// TwinCAT 3 PLC project ScriblyPlc
// ProgramVersion: 3.1.4023.0
// libraries:
//   Tc3_Module,3.3.21.0,Beckhoff Automation GmbH
//   Struckig, 0.9.0.0 (Stefan Besler)
//   ZApplication, 1.3.18.0 (Zeugwerk GmbH)
//   ZAux, 1.3.18.0 (Zeugwerk GmbH)
//   ZCore, 1.3.18.0 (Zeugwerk GmbH)
//   ZEquipment, 1.3.18.0 (Zeugwerk GmbH)
//   ZPlatform, 1.3.18.0 (Zeugwerk GmbH)
// project tree:
//   ZApp/App/ ZApp.TcPOU
//   ZApp/App/_DataTypes/ ZAppStep.TcDUT
//   ZApp/App/_States/ ZAppSequenceBoot.TcPOU, ZAppSequenceBootFault.TcPOU, ZAppSequenceRunning.TcPOU
//   ZApp/App/_SubObjects/ ZAppSequence.TcPOU
//   ZApp/Com/_DataTypes/ ZCom.TcDUT, ZComUnit.TcDUT
//   ZApp/Data/_DataTypes/ ZData.TcDUT, ZDataMachine.TcDUT, ZDataConfig.TcDUT, ZDataCalibration.TcDUT, ZDataRecipe.TcDUT
//   ZApp/Unit/Scribly/ IScribly.TcIO, ScriblyUnit.TcPOU, ScriblyUnitProgram.TcPOU
//   ZApp/Unit/Scribly/Segments/ RingBufferSegment.TcPOU, Segment.TcDUT, SegmentType.TcDUT
//   ZApp/Unit/Scribly/_Com/ ScriblyCom.TcDUT, ScriblyComPublish.TcDUT, ScriblyComPublishEquipment.TcDUT, ScriblyComRef.TcDUT, ScriblyComRequest.TcDUT, ScriblyComSubscribe.TcDUT, ScriblyComSubscribeEquipment.TcDUT, ScriblyComSubscribeSegments.TcDUT
//   ZApp/Unit/Scribly/_DataTypes/ ScriblyState.TcDUT, ScriblyStep.TcDUT
//   ZApp/Unit/Scribly/_Data/ ScriblyDataCalibration.TcDUT, ScriblyDataConfig.TcDUT, ScriblyDataMachine.TcDUT, ScriblyDataRef.TcDUT
//   ZApp/Unit/Scribly/_Equipment/ ScriblyActuator.TcPOU, ScriblyActuatorPen.TcPOU, ScriblyAxis.TcPOU, ScriblyEquipment.TcPOU, ScriblyFieldbus.TcPOU, ScriblyIo.TcPOU, ScriblyLinkedUnit.TcPOU
//   ZApp/Unit/Scribly/_States/ ScriblySequenceAutomatic.TcPOU, ScriblySequenceBoot.TcPOU, ScriblySequenceFaultReaction.TcPOU, ScriblySequenceGoHome.TcPOU, ScriblySequenceStop.TcPOU
//   ZApp/Unit/Scribly/_SubObjects/ ScriblyContainer.TcPOU, ScriblySequence.TcPOU
//   ZApp/ ZGlobal.TcGVL, ZModuleProgram.TcPOU, ZModuleTask.TcTTO
// real-time tasks:
//   TASK ZModuleTask: cycle T#10ms, priority 20, ADS port 350

CONFIGURATION ScriblyPlc
    RESOURCE PLC ON TwinCAT3
        TASK ZModuleTask(INTERVAL := T#10ms, PRIORITY := 20);
        PROGRAM ZeugwerkFramework WITH ZModuleTask : ZeugwerkFramework;
        PROGRAM ZModuleProgram WITH ZModuleTask : ZModuleProgram;
    END_RESOURCE
END_CONFIGURATION

// ---- ZApp/App/_DataTypes/ZAppStep.TcDUT
{attribute 'qualified_only'}
{attribute 'to_string'}
TYPE ZAppStep :
(
  Undefined := 0
  
  ,BootBegin
  ,BootLoadDefaultData
  ,BootEnd
  ,BootFaultBegin
  ,BootFaultEnd 
  ,RunningBegin
  ,RunningEnd   
);
END_TYPE

// ---- ZApp/Com/_DataTypes/ZCom.TcDUT
TYPE ZCom :
STRUCT
  // module context
  App : ZApplication.ApplicationComPublish;
  Alarming : ZApplication.AlarmingCom;
  Messages : ZApplication.MessagingCom;
  
  // unit context
  Unit : ZComUnit;

END_STRUCT
END_TYPE

// ---- ZApp/Com/_DataTypes/ZComUnit.TcDUT
TYPE ZComUnit :
STRUCT
{region "Scribly"}
{IF NOT (defined (Scribly_disabled))}
  Scribly : ScriblyCom;
  {attribute 'ZId' := '61e5b130-0fef-4d8b-85dd-afb1efcde47c'}
{END_IF}
{endregion}
{attribute '__ZwPlcApplicationComUnitDeclaration__'} // Do not remove this attribute! It is used for code generation.
END_STRUCT
END_TYPE

// ---- ZApp/Data/_DataTypes/ZData.TcDUT
TYPE ZData :
STRUCT
  Config : ZDataConfig;
  Machine : ZDataMachine;
  Calibration : ZDataCalibration;
  Recipe : ZDataRecipe;
END_STRUCT
END_TYPE

// ---- ZApp/Data/_DataTypes/ZDataMachine.TcDUT
TYPE ZDataMachine :
STRUCT
{region "Scribly"}
{IF NOT (defined (Scribly_disabled))}
  Scribly : ScriblyDataMachine;
  {attribute 'ZId' := '61e5b130-0fef-4d8b-85dd-afb1efcde47c'}
{END_IF}
{endregion}
{attribute '__ZwPlcApplicationDataMachineDeclaration__'} // Do not remove this attribute! It is used for code generation.
END_STRUCT
END_TYPE

// ---- ZApp/Data/_DataTypes/ZDataConfig.TcDUT
TYPE ZDataConfig :
STRUCT
{region "Scribly"}
{IF NOT (defined (Scribly_disabled))}
  Scribly : ScriblyDataConfig;
  {attribute 'ZId' := '61e5b130-0fef-4d8b-85dd-afb1efcde47c'}
{END_IF}
{endregion}
{attribute '__ZwPlcApplicationDataConfigDeclaration__'} // Do not remove this attribute! It is used for code generation.
END_STRUCT
END_TYPE

// ---- ZApp/Data/_DataTypes/ZDataCalibration.TcDUT
TYPE ZDataCalibration :
STRUCT
{region "Scribly"}
{IF NOT (defined (Scribly_disabled))}
  Scribly : ScriblyDataCalibration;
  {attribute 'ZId' := '61e5b130-0fef-4d8b-85dd-afb1efcde47c'}
{END_IF}
{endregion}
{attribute '__ZwPlcApplicationDataCalibrationDeclaration__'} // Do not remove this attribute! It is used for code generation.
END_STRUCT
END_TYPE

// ---- ZApp/Data/_DataTypes/ZDataRecipe.TcDUT
TYPE ZDataRecipe :
STRUCT
  RecipeParam1 : LREAL;
  RecipeParam2 : LREAL;
  RecipeParam3 : LREAL;
END_STRUCT
END_TYPE

// ---- ZApp/Unit/Scribly/Segments/Segment.TcDUT
TYPE Segment :
STRUCT
  Verb : SegmentType;
  Points : ARRAY[0..7] OF ZCore.Vector4;
END_STRUCT
END_TYPE

// ---- ZApp/Unit/Scribly/Segments/SegmentType.TcDUT
{attribute 'qualified_only'}
{attribute 'strict'}
TYPE SegmentType :
(
	Location := 0,
  LinePoints,
  CatmulRomPoints
);
END_TYPE

// ---- ZApp/Unit/Scribly/_Com/ScriblyCom.TcDUT
/// This struct contains variables that
/// * are read from outside (e.g. HMI) to retrieve information about the unit's current state and (temporary) parameters (= `publish`) 
/// * are written from outside (e.g. HMI) to control the unit via ADS (= `subscribe`) 
TYPE ScriblyCom :
STRUCT
  Publish : ScriblyComPublish;
  Subscribe : ScriblyComSubscribe;
END_STRUCT
END_TYPE

// ---- ZApp/Unit/Scribly/_Com/ScriblyComPublish.TcDUT
/// this is the container of informations that the unit wants to share with the world outside of the PLC
/// This struct should only be read from by external applications.
TYPE ScriblyComPublish :
STRUCT
  State : ZApplication.UnitStateMachineState; // state the unit is in
  Request : ScriblyComRequest; // booleans that indictate which action is currently possible to perform with this unit
  Equipment : ScriblyComPublishEquipment;  // structs for equipment objects which are used by the bridges
END_STRUCT
END_TYPE

// ---- ZApp/Unit/Scribly/_Com/ScriblyComPublishEquipment.TcDUT
TYPE ScriblyComPublishEquipment :
STRUCT

{region "Pen : ActuatorDigital"}
  Pen : ZApplication.ActuatorDigitalComPublish;
  PenDown : ZApplication.DigitalComPublish;
  PenUp : ZApplication.DigitalComPublish;
  PenIsDown : ZApplication.DigitalComPublish;
  PenIsUp : ZApplication.DigitalComPublish;
  {attribute 'ZId' := '715ceec0-4c65-4cb8-884b-f54d8c494ea5'}
{endregion}

{region "AxisX : Axis"}
  AxisX : ZApplication.AxisComPublish;
  {attribute 'ZId' := 'a9303431-20fb-4f90-9643-84006bcd2555'}
{endregion}

{region "AxisY : Axis"}
  AxisY : ZApplication.AxisComPublish;
  {attribute 'ZId' := '787e5d02-9d93-4b03-8235-ee23b1a291ad'}
{endregion}

{attribute '__ZwPlcUnitComDeclaration__'} // Do not remove this attribute! It is used for code generation.

END_STRUCT
END_TYPE

// ---- ZApp/Unit/Scribly/_Com/ScriblyComRef.TcDUT
/// container for all communication data types that are used by the unit
TYPE ScriblyComRef :
STRUCT
  Publish : REFERENCE TO ScriblyComPublish; 
  Subscribe : REFERENCE TO ScriblyComSubscribe; 
END_STRUCT
END_TYPE

// ---- ZApp/Unit/Scribly/_Com/ScriblyComRequest.TcDUT
TYPE ScriblyComRequest :
STRUCT
  Start : BOOL;
  Stop : BOOL;
  GoHome : BOOL;
  Halt : BOOL;
END_STRUCT
END_TYPE

// ---- ZApp/Unit/Scribly/_Com/ScriblyComSubscribe.TcDUT
TYPE ScriblyComSubscribe :
STRUCT
  Request : ScriblyComRequest; // contains booleans that are used to start a specific sequence.
  Equipment : ScriblyComSubscribeEquipment;  // structs for equipment objects which are used by the bridges
  
  Segments : ScriblyComSubscribeSegments;
END_STRUCT
END_TYPE

// ---- ZApp/Unit/Scribly/_Com/ScriblyComSubscribeEquipment.TcDUT
TYPE ScriblyComSubscribeEquipment :
STRUCT

{region "Pen : ActuatorDigital"}
  Pen : ZApplication.ActuatorDigitalComSubscribe;
  PenDown : ZApplication.DigitalComSubscribe;
  PenUp : ZApplication.DigitalComSubscribe;
  PenIsDown : ZApplication.DigitalComSubscribe;
  PenIsUp : ZApplication.DigitalComSubscribe;
  {attribute 'ZId' := '715ceec0-4c65-4cb8-884b-f54d8c494ea5'}
{endregion}

{region "AxisX : Axis"}
  AxisX : ZApplication.AxisComSubscribe;
  {attribute 'ZId' := 'a9303431-20fb-4f90-9643-84006bcd2555'}
{endregion}

{region "AxisY : Axis"}
  AxisY : ZApplication.AxisComSubscribe;
  {attribute 'ZId' := '787e5d02-9d93-4b03-8235-ee23b1a291ad'}
{endregion}

{attribute '__ZwPlcUnitComDeclaration__'} // Do not remove this attribute! It is used for code generation.

END_STRUCT
END_TYPE

// ---- ZApp/Unit/Scribly/_Com/ScriblyComSubscribeSegments.TcDUT
TYPE ScriblyComSubscribeSegments :
STRUCT
  Start : DINT;
  End : DINT;
  Data : ARRAY[0..10] OF Segment;
END_STRUCT
END_TYPE

// ---- ZApp/Unit/Scribly/_DataTypes/ScriblyState.TcDUT
/// This enumeration contains all used defined sequences of a unit.
/// Per default a unit makes use of the states that are contained in (UnitStateDefault)[xref:ZApplication.UnitStateDefault]. However,
/// most of the time a unit need to perform some application depend sequences that can be performed by putting the unit into userdefined states.
/// For instance, a robotic unit could use the state (automatic)[xref:ZApplication.UnitStateDefault] to lift an object from point A to point B,
/// a userdefined state could be used to open and close the robotic-units gripper, respectively
{attribute 'qualified_only'}
TYPE ScriblyState :
(
	UserdefinedState1 := ZApplication.UnitStateMachineState.Last+1
);
END_TYPE

// ---- ZApp/Unit/Scribly/_DataTypes/ScriblyStep.TcDUT
/// This enumeration contains all steps that are used by the various sequences of a unit.
/// Sequences use a subrange (***Begin to ***End) of this enumeration.
{attribute 'qualified_only'}
{attribute 'to_string'}
TYPE ScriblyStep :
(
  Undefined := 0
  
  ,BootBegin
  ,BootEnd 

  ,StopBegin
  ,StopEnd

  ,AutomaticBegin
  ,AutomaticWaitSegment
  ,AutomaticMoveToSegmentStart
  ,AutomaticMovePenDown
  ,AutomaticDraw
  ,AutomaticMovePenUp
  ,AutomaticDrawLine
  ,AutomaticDrawCatmulRomDrawSplineBegin
  ,AutomaticDrawCatmulRomDrawSpline
  ,AutomaticEnd
  
  ,GoHomeBegin
  ,GoHomeMoveUp  
  ,GoHomeReferenceXY
  ,GoHomeEnd 
  
  ,FaultReactionBegin
  ,FaultReactionEnd
);
END_TYPE

// ---- ZApp/Unit/Scribly/_Data/ScriblyDataCalibration.TcDUT
/// calibration that is determined by calibration sequences of the unit (static offsets, shifts)
TYPE ScriblyDataCalibration :
STRUCT
END_STRUCT
END_TYPE

// ---- ZApp/Unit/Scribly/_Data/ScriblyDataConfig.TcDUT
/// configuration data that is used during boot to configure the Units equipment
TYPE ScriblyDataConfig :
STRUCT
  Simulated : BOOL;
END_STRUCT
END_TYPE

// ---- ZApp/Unit/Scribly/_Data/ScriblyDataMachine.TcDUT
/// machine data that is used through most sequences of the unit (motor speed, axes positions, ...)
TYPE ScriblyDataMachine :
STRUCT
  Slowspeed : LREAL;
  Highspeed : LREAL;
END_STRUCT
END_TYPE

// ---- ZApp/Unit/Scribly/_Data/ScriblyDataRef.TcDUT
/// container for all data that are used by the unit
TYPE ScriblyDataRef :
STRUCT
  Config : REFERENCE TO ScriblyDataConfig; // data required for booting the unit (axes configuration, simulation, parameters that have to be written in PREOP, ...)
  Machine : REFERENCE TO ScriblyDataMachine; // speeds, positions, ...
  Calibration : REFERENCE TO ScriblyDataCalibration; // offsets, shifts of nominal to actual values
END_STRUCT
END_TYPE

// ---- ZApp/ZGlobal.TcGVL
{attribute 'qualified_only'}
VAR_GLOBAL
  Com : ZCom;
END_VAR
VAR_GLOBAL PERSISTENT
  Data : ZData;
END_VAR

// ---- ZApp/Unit/Scribly/IScribly.TcIO
INTERFACE IScribly EXTENDS ZApplication.IUnit

END_INTERFACE

// ---- ZApp/ZModuleProgram.TcPOU
/// Zeugwerk Application
PROGRAM ZModuleProgram
VAR
{region "ZModuleProgram : Utility"}
  App : ZApp(name:='Scribly', com:=ZGlobal.Com.App);
  Datetime : ZAux.DateTimeUM;
  {attribute 'ZId' := ''}
{endregion}
{region "ZModuleProgram : Logging"}
  Alarming : ZApplication.Alarming(App, datetime := Datetime, com := ZGlobal.Com.Alarming);
  LoggerHmi : ZApplication.Messaging(App, datetime := Datetime, com := ZGlobal.Com.Messages);
  LoggerFile : ZAux.LoggerFile7FF(App, datetime := Datetime, filePath:='C:\Zeugwerk\logs\messages.log', target:='');
  Logger : ZAux.Logging;
  {attribute 'ZId' := ''}
{endregion}  
{attribute '__ZwPlcApplicationModuleProgramDeclaration__'} // Do not remove this attribute! It is used for code generation.
{region "Scribly"}
{undefine RunInSeparateProgram}
{IF NOT (defined (Scribly_disabled)) AND NOT (defined (RunInSeparateProgram))}
  Scribly : ScriblyUnit(name := 'Scribly', // name of the unit (for logging)
					  parent := App, // caller of the Unit's cyclic method. If the Unit runs in its own context use 0
						configdata := ZGlobal.Data.Config.Scribly,
						machinedata := ZGlobal.Data.Machine.Scribly,
						calibrationdata := ZGlobal.Data.Calibration.Scribly,
						com := ZGlobal.Com.Unit.Scribly);
  {attribute 'section' := '__ZwPlcUnitProgramDeclaration__'}
  {attribute 'ZId' := '61e5b130-0fef-4d8b-85dd-afb1efcde47c'}
{END_IF}
{endregion}
{attribute '__ZwPlcUnitProgramDeclaration__'} // Do not remove this attribute! It is used for code generation.
END_VAR

{region "ZModuleProgram : Utility"}
  Datetime.Cyclic();
  App.Cyclic();
  {attribute 'ZId' := ''}
{endregion}
{attribute '__ZwPlcApplicationModuleProgramImplementation__'} // Do not remove this attribute! It is used for code generation.

END_PROGRAM

// ---- ZApp/App/ZApp.TcPOU
FUNCTION_BLOCK ZApp EXTENDS ZApplication.Application
VAR
  _boot : ZAppSequenceBoot;
  _bootFault : ZAppSequenceBootFault;
  _running : ZAppSequenceRunning;
END_VAR

METHOD FB_init : BOOL
VAR_INPUT
  bInitRetains : BOOL; /// if TRUE, the retain variables are initialized (warm start / cold start)
  bInCopyCode : BOOL; /// if TRUE, the instance afterwards gets moved into the copy code (online change)
  name : ZCore.ZString;
  com : REFERENCE TO ZApplication.ApplicationComPublish;
END_VAR
SetBootSequence(_boot);
SetBootFaultSequence(_bootFault);
SetRunningSequence(_running);
END_METHOD

END_FUNCTION_BLOCK

// ---- ZApp/App/_States/ZAppSequenceBoot.TcPOU
FUNCTION_BLOCK ZAppSequenceBoot EXTENDS ZAppSequence IMPLEMENTS ZCore.ISequence
VAR
  _step : ZCore.Step(ZAppStep.BootBegin, ZAppStep.BootEnd);
END_VAR

IF OnStart(_step)
THEN
  // init custom sequence variables here ...
END_IF

REPEAT
  LogStep();

  CASE _step.Index OF
    (* -------------------------------------------------------------------------------------------------------------------------------- *)
    ZAppStep.BootBegin:
    (* -------------------------------------------------------------------------------------------------------------------------------- *)
    
      IF _step.OnEntry()
      THEN
        ZModuleProgram.LoggerFile.SetLevel(ZCore.LogLevel.Trace);
        ZModuleProgram.Logger.AddLogger(ZModuleProgram.LoggerFile);        
        {attribute '__ZwPlcAppZComModuleContext__'} // Do not remove this attribute! It is used for code generation.      
      END_IF
      
	  IF ZModuleProgram.Datetime.State <> ZCore.ObjectState.Booting
      THEN
        _step.SetNext(ZAppStep.BootLoadDefaultData);        
      END_IF
      
    (* -------------------------------------------------------------------------------------------------------------------------------- *)
    ZAppStep.BootLoadDefaultData:
    (* -------------------------------------------------------------------------------------------------------------------------------- *)

      {warning 'The application is loading the default config data on every restart!'}
      LoadDefaultConfigData();
      
      IF IsCommissioning()
      THEN
        LoadDefaultData();
      END_IF
      
      _step.SetNext(ZAppStep.BootEnd);
      
    (* -------------------------------------------------------------------------------------------------------------------------------- *)
    ZAppStep.BootEnd:
    (* -------------------------------------------------------------------------------------------------------------------------------- *)
      SetBusy(FALSE);
      
  ELSE
    Abort('sequence contains unhandled step');
  END_CASE
UNTIL _step.IsNotRepeatable() OR_ELSE NOT Busy END_REPEAT

METHOD  IsCommissioning : BOOL
IsCommissioning := TRUE;
END_METHOD

METHOD FINAL LoadDefaultConfigData

{region "Scribly"}
  {IF NOT (defined (Scribly_disabled))}
  ZGlobal.Data.Config.Scribly.Simulated := TRUE;
  {region "UserInitCode"}
  // put your individual init code for this unit here
  {endregion}
  {END_IF}
  {attribute 'ZId' := '61e5b130-0fef-4d8b-85dd-afb1efcde47c'}
{endregion}

{attribute '__ZwPlcUnitLoadDefaultConfigData__'} // Do not remove this attribute! It is used for code generation.
END_METHOD

METHOD FINAL LoadDefaultData

{attribute '__ZwPlcUnitLoadDefaultData__'} // Do not remove this attribute! It is used for code generation.
ZGlobal.Data.Machine.Scribly.Highspeed := 100;
ZGlobal.Data.Machine.Scribly.Slowspeed := 10;
END_METHOD

END_FUNCTION_BLOCK

// ---- ZApp/App/_SubObjects/ZAppSequence.TcPOU
FUNCTION_BLOCK ABSTRACT ZAppSequence EXTENDS ZApplication.Sequence IMPLEMENTS ZCore.ISequence

METHOD StepDecoded : ZCore.ZString
VAR_INPUT
  stepIndex : INT;
END_VAR
VAR_INST
  _stepIndexDecoded : ZAppStep;
END_VAR
_stepIndexDecoded := stepIndex;
StepDecoded := TO_STRING(_stepIndexDecoded);
END_METHOD

END_FUNCTION_BLOCK

// ---- ZApp/App/_States/ZAppSequenceBootFault.TcPOU
FUNCTION_BLOCK ZAppSequenceBootFault EXTENDS ZAppSequence IMPLEMENTS ZCore.ISequence
VAR
  _step : ZCore.Step(ZAppStep.BootFaultBegin, ZAppStep.BootFaultEnd);
END_VAR

IF OnStart(_step)
THEN
  // init custom sequence variables here ...
END_IF

REPEAT
  LogStep();

  CASE _step.Index OF
    (* -------------------------------------------------------------------------------------------------------------------------------- *)
    ZAppStep.BootFaultBegin:
    (* -------------------------------------------------------------------------------------------------------------------------------- *)
      _step.SetNext(ZAppStep.BootFaultEnd);
      
    (* -------------------------------------------------------------------------------------------------------------------------------- *)
    ZAppStep.BootFaultEnd:
    (* -------------------------------------------------------------------------------------------------------------------------------- *)
      SetBusy(FALSE);
      
  ELSE
    Abort('sequence contains unhandled step');
  END_CASE
UNTIL _step.IsNotRepeatable() OR_ELSE NOT Busy END_REPEAT

END_FUNCTION_BLOCK

// ---- ZApp/App/_States/ZAppSequenceRunning.TcPOU
FUNCTION_BLOCK ZAppSequenceRunning EXTENDS ZAppSequence IMPLEMENTS ZCore.ISequence
VAR
  _step : ZCore.Step(ZAppStep.RunningBegin, ZAppStep.RunningEnd);
END_VAR

IF OnStart(_step)
THEN
  // init custom sequence variables here ...
END_IF

REPEAT
  LogStep();

  CASE _step.Index OF
    (* -------------------------------------------------------------------------------------------------------------------------------- *)
    ZAppStep.RunningBegin:
    (* -------------------------------------------------------------------------------------------------------------------------------- *)
      ; // implement me
      
    (* -------------------------------------------------------------------------------------------------------------------------------- *)
    ZAppStep.RunningEnd:
    (* -------------------------------------------------------------------------------------------------------------------------------- *)
      SetBusy(FALSE);
      
  ELSE
    Abort('sequence contains unhandled step');
  END_CASE
UNTIL _step.IsNotRepeatable() OR_ELSE NOT Busy END_REPEAT

END_FUNCTION_BLOCK

// ---- ZApp/Unit/Scribly/ScriblyUnit.TcPOU
/// Declaration of a distinct unit of this application
FUNCTION_BLOCK ScriblyUnit EXTENDS ZApplication.Unit IMPLEMENTS IScribly, ZAux.IStateMachineListener
VAR
  _equipment : ScriblyEquipment(THIS^);
  _data : ScriblyDataRef;
  _com : ScriblyComRef;

  _boot : ScriblySequenceBoot(THIS^);
  _automatic : ScriblySequenceAutomatic(THIS^);
  _stop : ScriblySequenceStop(THIS^);
  _gohome : ScriblySequenceGoHome(THIS^);
  _faultReaction : ScriblySequenceFaultReaction(THIS^);
  
  _statemachine : ZApplication.UnitStateMachine;

  _observeTimer : ZAux.Timer;
  _segments : RingBufferSegment(
                10, 
                ADR(ZGlobal.Com.Unit.Scribly.Subscribe.Segments.Start),
                ADR(ZGlobal.Com.Unit.Scribly.Subscribe.Segments.End),
                ADR(ZGlobal.Com.Unit.Scribly.Subscribe.Segments.Data));        
END_VAR

{attribute 'ZId' := 'f607484c-b594-4144-a307-86b8991e3218'}

IF _observeTimer.Done THEN
  _observeTimer.WaitAsync(0.1);
  
  // monitor _com for requested actions (e.g. start homing, start automatic mode, ...)
  ObserveRequest(_com.Subscribe.Request.Start, ZApplication.UnitStateMachineState.Automatic);
  ObserveRequest(_com.Subscribe.Request.Stop, ZApplication.UnitStateMachineState.Stop);
  ObserveRequest(_com.Subscribe.Request.GoHome, ZApplication.UnitStateMachineState.GoHome);
  ObserveRequest(_com.Subscribe.Request.Halt, ZApplication.UnitStateMachineState.Halt);
  
  // provide relevant information via ADS
  _com.Publish.Request.Stop := _stateMachine.IsTransitionAllowed(ZApplication.UnitStateMachineState.Stop);
  _com.Publish.Request.Start := _stateMachine.IsTransitionAllowed(ZApplication.UnitStateMachineState.Automatic);
  _com.Publish.Request.GoHome := _stateMachine.IsTransitionAllowed(ZApplication.UnitStateMachineState.GoHome);
  _com.Publish.Request.Halt := _stateMachine.IsTransitionAllowed(ZApplication.UnitStateMachineState.Halt);

  _com.Publish.State := _stateMachine.State();
END_IF

METHOD FB_init : BOOL
VAR_INPUT
  bInitRetains : BOOL; // if TRUE, the retain variables are initialized (warm start / cold start)
  bInCopyCode : BOOL;  // if TRUE, the instance afterwards gets moved into the copy code (online change)
  parent : ZCore.IManagedObject; // caller of the Unit's cyclic method. If the Unit runs in its own context use 0
  name : ZCore.ZString;  // name of this unit as it should show up in the logger
  configdata : REFERENCE TO ScriblyDataConfig;  // reference to the configuration data that is used during boot to configure the Units equipment
  machinedata : REFERENCE TO ScriblyDataMachine; // reference to the machine data that is used through most sequences of the unit (motor speed, axes positions, ...)
  calibrationdata : REFERENCE TO ScriblyDataCalibration;  // reference to calibration that is determined by calibration sequences of the unit (static offsets, shifts)
  com : REFERENCE TO ScriblyCom;  // reference to the communication interface that is used to control this Unit via ADS
END_VAR
_name := name;

// initialize local logger decorator
_loggerDecorator.FB_init(bInitRetains, bInCopyCode, name, ZModuleProgram.Logger);
_alarmingDecorator.FB_init(bInitRetains, bInCopyCode, name, ZModuleProgram.Alarming);

// setup data
_data.Config REF= configdata;
_data.Machine REF= machinedata;
_data.Calibration REF= calibrationdata;
_com.Publish REF= com.Publish;
_com.Subscribe REF= com.Subscribe;

// ------- sequence initialization, map sequences of this unit to the statemachine -------
{attribute '__ZwPlcUnitInitSequenceImplementation__'} // Do not remove this attribute! It is used for code generation.
_statemachine.SetSequence(ZApplication.UnitStateMachineState.Boot, _boot);
_statemachine.SetSequence(ZApplication.UnitStateMachineState.FaultReaction, _faultReaction);
_statemachine.SetSequence(ZApplication.UnitStateMachineState.Gohome, _gohome);
_statemachine.SetSequence(ZApplication.UnitStateMachineState.Stop, _stop);
_statemachine.SetSequence(ZApplication.UnitStateMachineState.Automatic, _automatic);

_statemachine.SetName(_name);
_statemachine.SetListener(THIS^);
_statemachine.SetLogger(_logger);

// set initial state
_statemachine.SetState(ZApplication.UnitStateMachineState.Boot);
_statemachineIntrf := _statemachine;
END_METHOD

/// This method is called by a [Statemachine's startTransition method](xref:ZApplication.UnitStateMachine#startTransition)
/// if a given transition was failed (e.g. the transition is not allowed according to the state diagram of the state machine).
/// The State that was active previously in the StateMachine remains active and `requestedState` indicates which state transition
/// was requested by the user.
METHOD OnStartTransitionFailed
VAR_INPUT
  state : INT;  
  requestedState : INT;
END_VAR
END_METHOD

/// This method is called by a [Statemachine's startTransition method](xref:ZApplication.UnitStateMachine#startTransition)
/// if a given transition was successful. Please note, that at the time this event occurs, `state` still holds the
/// state that was active before calling `startTransition`, there is still one more call to this `state` to allow it to 
/// cleanup.
METHOD OnStartTransitionSucceeded
VAR_INPUT
  state : INT;  
  newState : INT;
END_VAR
END_METHOD

/// This method is called after a transition succeeded, right before the [start method of a sequence](xref:ZAux#start) is called.
/// The parameter `state` indicates the State that is active in the statemachine.
METHOD OnStateEntry
VAR_INPUT
  state : INT;
END_VAR
END_METHOD

/// This method is called after a sequence reported an error, but before the state machine starts its error handling.
METHOD OnStateError
VAR_INPUT
  state : INT;
END_VAR
END_METHOD

/// This method is called after a transition succeeded, right before the [stop method of a sequence](xref:ZAux#start) is called.
/// The parameter `state` indicates the State that is active in the statemachine.
METHOD OnStateExit
VAR_INPUT
  state : INT;  
END_VAR
END_METHOD

/// This method if a State has been executed successfully.
/// The parameter `state` indicates the State that is active in the statemachine.
METHOD OnStateSuccess
VAR_INPUT
  state : INT;    
END_VAR
END_METHOD

END_FUNCTION_BLOCK

// ---- ZApp/Unit/Scribly/_Equipment/ScriblyEquipment.TcPOU
/// This function block is a container for equipment that is used by this unit.
/// Equipment is grouped by its kind (actuator, axes, io, ...).
/// It extends from [ManagedObjectContainer](xref:ZCore.ManagedObjectContainer) such that the parent
/// (= the unit itself) can be passed to equipment instances.
FUNCTION_BLOCK ScriblyEquipment EXTENDS ScriblyContainer
VAR_INPUT
  Io : ScriblyIo(_parent);
  Actuator : ScriblyActuator(_parent);
  Axis : ScriblyAxis(_parent);
  Fieldbus : ScriblyFieldbus(_parent);
  Unit : ScriblyLinkedUnit(_parent);
END_VAR

END_FUNCTION_BLOCK

// ---- ZApp/Unit/Scribly/_SubObjects/ScriblyContainer.TcPOU
FUNCTION_BLOCK ScriblyContainer EXTENDS ZCore.ObjectContainer
VAR_INPUT
END_VAR
VAR_OUTPUT
END_VAR
VAR
  {attribute 'hide'}
  _parent : REFERENCE TO ScriblyUnit;
END_VAR

{ attribute 'hide' }
METHOD FB_init : BOOL
VAR_INPUT
	bInitRetains : BOOL; // if TRUE, the retain variables are initialized (warm start / cold start)
	bInCopyCode : BOOL;  // if TRUE, the instance afterwards gets moved into the copy code (online change)
  unit : REFERENCE TO ScriblyUnit;
END_VAR
_parent REF= unit;
END_METHOD

END_FUNCTION_BLOCK

// ---- ZApp/Unit/Scribly/_Equipment/ScriblyIo.TcPOU
/// This function block is a container for all I/Os that are used by this unit.
/// The parent of all objects can be directly transfered in their constructor (this is only relevant for equipment objects
/// that have to be managed (e.g. [DebouncedInput](xref:ZEquipment.DebouncedInput), [Light](xref:ZEquipment.Light), ...).
FUNCTION_BLOCK ScriblyIo EXTENDS ScriblyContainer
VAR
  {attribute 'hide'}
  _iobridge : ZApplication.IoBridge(_parent);
END_VAR
VAR_INPUT

{attribute '__ZwPlcUnitEquipmentDeclaration__'} // Do not remove this attribute! It is used for code generation.
END_VAR

IF _isInitialized
THEN
  RETURN;
END_IF

  _iobridge.SetLogger(_parent._logger);

{attribute '__ZwPlcUnitEquipmentImplementation__'} // Do not remove this attribute! It is used for code generation.

_isInitialized := TRUE;

END_FUNCTION_BLOCK

// ---- ZApp/Unit/Scribly/_Equipment/ScriblyActuator.TcPOU
/// This function block is a container for all actuator objects that are used by this unit.
/// The parent of all objects can be directly transfered in their constructor (this is only relevant for equipment objects
/// that have to be managed (e.g. [DebouncedInput](xref:ZEquipment.DebouncedInput), [Light](xref:ZEquipment.Light), ...).
FUNCTION_BLOCK ScriblyActuator EXTENDS ScriblyContainer
VAR
  {attribute 'hide'}
  _actuatorbridge : ZApplication.ActuatorBridge(_parent);
  {attribute 'hide'}
  _iobridge : ZApplication.IoBridge(_parent);
END_VAR
VAR_INPUT

{region "Pen : ActuatorDigitalBiLsPlusMinus"}
  Pen : ScriblyActuatorPen(_parent);
  {attribute 'ZId' := '715ceec0-4c65-4cb8-884b-f54d8c494ea5'}
{endregion}

{attribute '__ZwPlcUnitEquipmentDeclaration__'} // Do not remove this attribute! It is used for code generation.
END_VAR

IF _isInitialized
THEN
  RETURN;
END_IF

  _actuatorbridge.SetLogger(_parent._logger);

{region "Pen : ActuatorDigitalBiLsPlusMinus"}
  Pen.SetLogger(_parent._logger);
  Pen.SetName(name:='Pen', movePlusName:='Up', moveMinusName:='Down', plusName:='IsUp', minusName:='IsDown');
  Pen.SetSimulation(SEL(_parent._data.Config.Simulated, ActuatorDigitalSimulation.Disabled, ZEquipment.ActuatorDigitalSimulation.Automatic));
  Pen.SetSimulationUncertainty(uncertainty:=10);
  Pen.SetDelay(plusStartDuration:=0, plusEndDuration:=0, minusStartDuration:=0, minusEndDuration:=0, stop:=0);
  Pen.SetSwitchDuration(plusDuration:=0.2, minusDuration:=0.2);
  Pen.SetMovementDuration(plusDuration:=3, minusDuration:=3);
  Pen.SetTimeout(plusDuration:=5, minusDuration:=5);
  _actuatorbridge.AddActuatorDigital(Pen, publish := _parent._com.Publish.Equipment.Pen, subscribe := _parent._com.Subscribe.Equipment.Pen);
  _iobridge.AddDigitalOutput(Pen.MinusOutput, publish := _parent._com.Publish.Equipment.PenDown, subscribe := _parent._com.Subscribe.Equipment.PenDown);
  _iobridge.AddDigitalOutput(Pen.PlusOutput, publish := _parent._com.Publish.Equipment.PenUp, subscribe := _parent._com.Subscribe.Equipment.PenUp);
  _iobridge.AddDigitalInput(Pen.MinusInput, publish := _parent._com.Publish.Equipment.PenIsDown, subscribe := _parent._com.Subscribe.Equipment.PenIsDown);
  _iobridge.AddDigitalInput(Pen.PlusInput, publish := _parent._com.Publish.Equipment.PenIsUp, subscribe := _parent._com.Subscribe.Equipment.PenIsUp);
  {region "UserInitCode"}
  // put your individual init code for this Actuator here
  {endregion}

  {attribute 'ZId' := '715ceec0-4c65-4cb8-884b-f54d8c494ea5'}
{endregion}

{attribute '__ZwPlcUnitEquipmentImplementation__'} // Do not remove this attribute! It is used for code generation.

_isInitialized := TRUE;

END_FUNCTION_BLOCK

// ---- ZApp/Unit/Scribly/_Equipment/ScriblyActuatorPen.TcPOU
FUNCTION_BLOCK ScriblyActuatorPen EXTENDS ZEquipment.ActuatorDigitalBiLsPlusMinus

METHOD PUBLIC DownAsync
VAR_INPUT
  startToken : ZCore.IStartToken;
END_VAR
MoveMinusAsync(startToken:=startToken);
END_METHOD

METHOD PUBLIC IsDown : BOOL
VAR_INPUT
END_VAR
IsDown := IsAtMinus();
END_METHOD

METHOD PUBLIC IsUp : BOOL
VAR_INPUT
END_VAR
IsUp := IsAtPlus();
END_METHOD

METHOD PUBLIC UpAsync
VAR_INPUT
  startToken : ZCore.IStartToken;
END_VAR
MovePlusAsync(startToken:=startToken);
END_METHOD

END_FUNCTION_BLOCK

// ---- ZApp/Unit/Scribly/_Equipment/ScriblyAxis.TcPOU
/// This function block is a container for all axis objects that are used by this unit.
/// The parent of all objects can be directly transfered in their constructor (this is only relevant for equipment objects
/// that have to be managed (e.g. [DebouncedInput](xref:ZEquipment.DebouncedInput), [Light](xref:ZEquipment.Light), ...).
FUNCTION_BLOCK ScriblyAxis EXTENDS ScriblyContainer
VAR
  {attribute 'hide'}
  _axisbridge : ZApplication.AxisBridge(_parent);
END_VAR
VAR_INPUT

{region "AxisX : AxisPlcOpenMc"}
  AxisX : ZEquipment.AxisPlcOpenMc(_parent);
  {attribute 'ZId' := 'a9303431-20fb-4f90-9643-84006bcd2555'}
{endregion}

{region "AxisY : AxisPlcOpenMc"}
  AxisY : ZEquipment.AxisPlcOpenMc(_parent);
  {attribute 'ZId' := '787e5d02-9d93-4b03-8235-ee23b1a291ad'}
{endregion}

{attribute '__ZwPlcUnitEquipmentDeclaration__'} // Do not remove this attribute! It is used for code generation.
END_VAR

IF _isInitialized
THEN
  RETURN;
END_IF

  _axisbridge.SetLogger(_parent._logger);

{region "AxisX : AxisPlcOpenMc"}
  AxisX.SetLogger(_parent._logger);
  AxisX.SetName(name:='AxisX');
  AxisX.SetSimulation(_parent._data.Config.Simulated);
  _axisbridge.AddAxisPlcOpenMc(axis:=AxisX, publish:=_parent._com.Publish.Equipment.AxisX, subscribe:=_parent._com.Subscribe.Equipment.AxisX);

  {region "UserInitCode"}
  // put your individual init code for this Axis here
  {endregion}

  {attribute 'ZId' := 'a9303431-20fb-4f90-9643-84006bcd2555'}
{endregion}

{region "AxisY : AxisPlcOpenMc"}
  AxisY.SetLogger(_parent._logger);
  AxisY.SetName(name:='AxisY');
  AxisY.SetSimulation(_parent._data.Config.Simulated);
  _axisbridge.AddAxisPlcOpenMc(axis:=AxisY, publish:=_parent._com.Publish.Equipment.AxisY, subscribe:=_parent._com.Subscribe.Equipment.AxisY);

  {region "UserInitCode"}
  // put your individual init code for this Axis here
  {endregion}

  {attribute 'ZId' := '787e5d02-9d93-4b03-8235-ee23b1a291ad'}
{endregion}

{attribute '__ZwPlcUnitEquipmentImplementation__'} // Do not remove this attribute! It is used for code generation.

_isInitialized := TRUE;

END_FUNCTION_BLOCK

// ---- ZApp/Unit/Scribly/_Equipment/ScriblyFieldbus.TcPOU
/// This function block is a container for all axis objects that are used by this unit.
/// The parent of all objects can be directly transfered in their constructor (this is only relevant for equipment objects
/// that have to be managed (e.g. [DebouncedInput](xref:ZEquipment.DebouncedInput), [Light](xref:ZEquipment.Light), ...).
FUNCTION_BLOCK ScriblyFieldbus EXTENDS ScriblyContainer
VAR
END_VAR
VAR_INPUT

{attribute '__ZwPlcUnitEquipmentDeclaration__'} // Do not remove this attribute! It is used for code generation.
END_VAR

IF _isInitialized
THEN
  RETURN;
END_IF

{attribute '__ZwPlcUnitEquipmentImplementation__'} // Do not remove this attribute! It is used for code generation.

_isInitialized := TRUE;

END_FUNCTION_BLOCK

// ---- ZApp/Unit/Scribly/_Equipment/ScriblyLinkedUnit.TcPOU
/// This function block is a container for all linked units that are used by this unit.
/// Linked units can be addressed through their individual interface.
FUNCTION_BLOCK ScriblyLinkedUnit EXTENDS ScriblyContainer
VAR_INPUT

{attribute '__ZwPlcUnitEquipmentDeclaration__'} // Do not remove this attribute! It is used for code generation.
END_VAR

IF _isInitialized
THEN
  RETURN;
END_IF

{attribute '__ZwPlcUnitEquipmentImplementation__'} // Do not remove this attribute! It is used for code generation.

_isInitialized := TRUE;

END_FUNCTION_BLOCK

// ---- ZApp/Unit/Scribly/_States/ScriblySequenceBoot.TcPOU
FUNCTION_BLOCK ScriblySequenceBoot EXTENDS ScriblySequence IMPLEMENTS ZCore.ISequence
VAR
  _step : ZCore.Step(ScriblyStep.BootBegin, ScriblyStep.BootEnd);
END_VAR

IF OnStart(_step) THEN
  ; // init custom sequence variables here ...
END_IF

REPEAT
  LogStep();

  CASE _step.Index OF
    (* -------------------------------------------------------------------------------------------------------------------------------- *)
    ScriblyStep.BootBegin:
    (* -------------------------------------------------------------------------------------------------------------------------------- *)
      IF _step.OnEntry()
      THEN
        // initialize equipment
        _io();
        _actuator();
        _fieldbus();
        _axis();
        _unit();
      END_IF
      
      _parent._objectManager.Cyclic();      
      Assert(_parent._objectManager);
      IF _parent._objectManager.Done
      THEN
        _step.SetNext(ScriblyStep.BootEnd);
      END_IF

    (* -------------------------------------------------------------------------------------------------------------------------------- *)
    ScriblyStep.BootEnd:
    (* -------------------------------------------------------------------------------------------------------------------------------- *)
      SetBusy(FALSE);
      
  ELSE
    Abort('sequence contains unhandled step');
  END_CASE
UNTIL _step.IsNotRepeatable() OR_ELSE NOT Busy END_REPEAT

END_FUNCTION_BLOCK

// ---- ZApp/Unit/Scribly/_SubObjects/ScriblySequence.TcPOU
FUNCTION_BLOCK ScriblySequence EXTENDS ZApplication.Sequence
VAR
  {attribute 'hide'}
  _parent : REFERENCE TO ScriblyUnit;
  _io : REFERENCE TO ScriblyIo;
  _actuator : REFERENCE TO ScriblyActuator;
  _fieldbus : REFERENCE TO ScriblyFieldbus;
  _axis : REFERENCE TO ScriblyAxis;
  _data : REFERENCE TO ScriblyDataRef;
  _unit : REFERENCE TO ScriblyLinkedUnit;
  _segments : REFERENCE TO RingBufferSegment;
END_VAR

METHOD FB_init : BOOL
VAR_INPUT
  bInitRetains : BOOL; // if TRUE, the retain variables are initialized (warm start / cold start)
  bInCopyCode : BOOL;  // if TRUE, the instance afterwards gets moved into the copy code (online change)
  unit : REFERENCE TO ScriblyUnit;
END_VAR
_parent REF= unit;
_alarming := unit._alarming;
_io REF= unit._equipment.Io;
_actuator REF= unit._equipment.Actuator;
_fieldbus REF= unit._equipment.Fieldbus;
_axis REF= unit._equipment.Axis;
_unit REF= unit._equipment.Unit;
_data REF= unit._data;
_loggerDiagnostics.SetLogger(unit._logger);

_segments REF= unit._segments;
END_METHOD

METHOD StepDecoded : ZCore.ZString
VAR_INPUT
  stepIndex : INT;
END_VAR
VAR_INST
  _stepIndexDecoded : ScriblyStep;
END_VAR
_stepIndexDecoded := stepIndex;
stepDecoded := TO_STRING(_stepIndexDecoded);
END_METHOD

END_FUNCTION_BLOCK

// ---- ZApp/Unit/Scribly/Segments/RingBufferSegment.TcPOU
FUNCTION_BLOCK RingBufferSegment EXTENDS ZCore.RingBuffer
VAR
  _dataPtr : POINTER TO Segment;  
END_VAR

/// Initializes the RingBuffer at construction time of the object by providing the bufferSize.
/// It also inidializes the pointers of head and tail with an internally stored variable.
METHOD FB_init : BOOL
VAR_INPUT
  bInitRetains : BOOL; //< if TRUE, the retain variables are initialized (warm start / cold start)
  bInCopyCode : BOOL; //< if TRUE, the instance afterwards gets moved into the copy code (online change)
  bufferSize : DINT; //< size of the **managable** buffer. The actual databuffer needs to be one element larger than bufferSize, i.e. data : ARRAY[0..bufferSize] OF ???
  startPtr : POINTER TO DINT;
  endPtr : POINTER TO DINT;
  dataPtr : POINTER TO Segment;
END_VAR
SetLogicPtrs(startPtr, endPtr);
_dataPtr := dataPtr;
END_METHOD

METHOD ItemAt : REFERENCE TO Segment
VAR_INPUT
  pos : DINT;
END_VAR
ItemAt REF= _dataPtr[IndexOfItem(pos)];
END_METHOD

END_FUNCTION_BLOCK

// ---- ZApp/Unit/Scribly/_States/ScriblySequenceAutomatic.TcPOU
FUNCTION_BLOCK ScriblySequenceAutomatic EXTENDS ScriblySequence IMPLEMENTS ZCore.ISequence
VAR
  _step : ZCore.Step(ScriblyStep.AutomaticBegin, ScriblyStep.AutomaticEnd);
  _segment : REFERENCE TO Segment;
  _rt : ZAux.RealTime;
  _otg : Struckig.Otg(0.001, 2);
  
  _splineLogicBuffer : ARRAY [0..8] OF DINT;
  _splinePointBuffer : ARRAY [0..8*2] OF LREAL;
  _splineTangentBuffer : ARRAY [0..8*2] OF LREAL;
  _splineSegmentBuffer : ARRAY [0..8] OF LREAL;
  _spline : ZCore.CatmullRomSpline(8, ADR(_splineLogicBuffer), ADR(_splinePointBuffer), ADR(_splineTangentBuffer), ADR(_splineSegmentBuffer), 2);
  
  _splineIndex : INT;
  i : INT;
END_VAR
VAR_OUTPUT
  ProbeX : LREAL;
  ProbeY : LREAL;
END_VAR

IF NOT Busy THEN
  RETURN;
END_IF

IF OnStart(_step) THEN
  ; // init custom sequence variables here ...
END_IF

IF OnStop() THEN
  RETURN; // external stop was triggered
END_IF

IF OnHalt() THEN
  Halting := TRUE; // Uncomment to acknowledge that the sequence is halting
END_IF

REPEAT
  LogStep();

  CASE _step.Index OF
    (* -------------------------------------------------------------------------------------------------------------------------------- *)
    ScriblyStep.AutomaticBegin:
    (* -------------------------------------------------------------------------------------------------------------------------------- *)
      IF _step.OnEntry()
      THEN
        ;
      END_IF

      _step.SetNext(ScriblyStep.AutomaticWaitSegment);
    
    (* -------------------------------------------------------------------------------------------------------------------------------- *)
    ScriblyStep.AutomaticWaitSegment:
    (* -------------------------------------------------------------------------------------------------------------------------------- *)
      IF _step.OnEntry()
      THEN
        Milestone('Waiting for segment');
      END_IF

      IF Halting
      THEN
        _step.SetNext(ScriblyStep.AutomaticEnd);
      ELSIF NOT _segments.Empty
      THEN
        _segment REF= _segments.ItemAt(0);
        _step.SetNext(ScriblyStep.AutomaticMoveToSegmentStart);
			END_IF


    (* -------------------------------------------------------------------------------------------------------------------------------- *)
    ScriblyStep.AutomaticMoveToSegmentStart:
    (* -------------------------------------------------------------------------------------------------------------------------------- *)
      IF _step.OnEntry()
      THEN
        _axis.AxisX.MoveAbsoluteAsync(THIS^, _segment.Points[0].X, _data.Machine.Highspeed);
        _axis.AxisY.MoveAbsoluteAsync(THIS^, _segment.Points[0].Y, _data.Machine.Highspeed);        
      END_IF

      Await2(_axis.AxisX, _axis.AxisY, ScriblyStep.AutomaticMovePenDown);
    
    
    (* -------------------------------------------------------------------------------------------------------------------------------- *)
    ScriblyStep.AutomaticMovePenDown:
    (* -------------------------------------------------------------------------------------------------------------------------------- *)
      IF _step.OnEntry()
      THEN
        _actuator.Pen.DownAsync(THIS^);       
      END_IF

      Await(_actuator.Pen, ScriblyStep.AutomaticDraw);

    (* -------------------------------------------------------------------------------------------------------------------------------- *)
    ScriblyStep.AutomaticDraw:
    (* -------------------------------------------------------------------------------------------------------------------------------- *)
      
      CASE _segment.Verb
      OF
        SegmentType.LinePoints: _step.SetNext(ScriblyStep.AutomaticDrawLine);
        SegmentType.CatmulRomPoints: _step.SetNext(ScriblyStep.AutomaticDrawCatmulRomDrawSplineBegin);
      ELSE
        Abort('Unsupported Verb');     
			END_CASE
      
    (* -------------------------------------------------------------------------------------------------------------------------------- *)
    ScriblyStep.AutomaticMovePenUp:
    (* -------------------------------------------------------------------------------------------------------------------------------- *)
      IF _step.OnEntry()
      THEN
        _actuator.Pen.UpAsync(THIS^);
        _segments.PopFirstItem();
      END_IF

      Await(_actuator.Pen, ScriblyStep.AutomaticWaitSegment);
      
    (* -------------------------------------------------------------------------------------------------------------------------------- *)
    ScriblyStep.AutomaticDrawLine:
    (* -------------------------------------------------------------------------------------------------------------------------------- *)
      IF _step.OnEntry()
      THEN
        _otg.CycleTime := _rt.CycleTimeInSeconds();
        _otg.ControlInterface := Struckig.ControlInterfaceType.Position;
        _otg.CurrentAcceleration[0] := 0;
        _otg.CurrentAcceleration[1] := 0;
        _otg.CurrentVelocity[0] := 0;
        _otg.CurrentVelocity[1] := 0;        
        _otg.CurrentPosition[0] := _segment.Points[0].X;
        _otg.CurrentPosition[1] := _segment.Points[0].Y;
        _otg.Discretization := Struckig.DiscretizationType.Discrete;
        _otg.EnableAutoPropagate := TRUE;
        _otg.MaxJerk[0] := 100000;
        _otg.MaxJerk[1] := 100000;         
        _otg.MaxAcceleration[0] := 10000;
        _otg.MaxAcceleration[1] := 10000; 
        _otg.MaxVelocity[0] := 50;
        _otg.MaxVelocity[1] := 50;      
        _otg.Synchronization := Struckig.SynchronizationType.Phase;
        _otg.TargetPosition[0] := _segment.Points[1].X;
        _otg.TargetPosition[1] := _segment.Points[1].Y;        
        _otg.TargetAcceleration[0] := 0;
        _otg.TargetAcceleration[1] := 0;
        _otg.TargetVelocity[0] := 0;
        _otg.TargetVelocity[1] := 0;
      END_IF
      
      _otg();
      ProbeX := _otg.CurrentPosition[0];
      ProbeY := _otg.CurrentPosition[1];
      
      IF _otg.State = Struckig.TrajectoryState.Error
      THEN
        AbortErrorId(ANY_TO_UDINT(_otg.ErrorCode()), 'Trajectory Error');
      ELSIF _otg.State = Struckig.TrajectoryState.Idle
      THEN
        _step.SetNext(ScriblyStep.AutomaticMovePenUp);        
			END_IF

    (* -------------------------------------------------------------------------------------------------------------------------------- *)
    ScriblyStep.AutomaticDrawCatmulRomDrawSplineBegin:
    (* -------------------------------------------------------------------------------------------------------------------------------- *)
    
      _otg.CycleTime := _rt.CycleTimeInSeconds();
      _otg.ControlInterface := Struckig.ControlInterfaceType.Position;
      _otg.Discretization := Struckig.DiscretizationType.Discrete;
      _otg.EnableAutoPropagate := TRUE;
      _otg.MaxJerk[0] := 100000;
      _otg.MaxJerk[1] := 100000;         
      _otg.MaxAcceleration[0] := 10000;
      _otg.MaxAcceleration[1] := 10000; 
      _otg.MaxVelocity[0] := 50;
      _otg.MaxVelocity[1] := 50; 
      _otg.Synchronization := Struckig.SynchronizationType.Phase;    
      _otg.CurrentAcceleration[0] := 0;
      _otg.CurrentAcceleration[1] := 0;        
      _otg.CurrentVelocity[0] := 0;
      _otg.CurrentVelocity[1] := 0;        
      _otg.CurrentPosition[0] := _segment.Points[0].X;
      _otg.CurrentPosition[1] := _segment.Points[0].Y;
      _otg.TargetAcceleration[0] := 0;
      _otg.TargetAcceleration[1] := 0;  
      _spline.Clear();
      
      // todo: make this more dynamic ...
      FOR i:=1 TO 8
      DO 
        _spline.Append3((i-1) / INT_TO_LREAL(7), _segment.Points[i].X, _segment.Points[i].Y, _segment.Points[i].Z);
      END_FOR

      _splineIndex := 0;
      _step.SetNext(ScriblyStep.AutomaticDrawCatmulRomDrawSpline);
      

    (* -------------------------------------------------------------------------------------------------------------------------------- *)
    ScriblyStep.AutomaticDrawCatmulRomDrawSpline:
    (* -------------------------------------------------------------------------------------------------------------------------------- *)
      IF _step.OnEntry()
      THEN
        _otg.TargetPosition[0] := _splinePointBuffer[_splineIndex*2];
        _otg.TargetPosition[1] := _splinePointBuffer[_splineIndex*2+1];      
        _otg.TargetVelocity[0] := _splineTangentBuffer[_splineIndex*2+1]; 
        _otg.TargetVelocity[1] := _splineTangentBuffer[_splineIndex*2+1]; 
      END_IF
      
      _otg();
      ProbeX := _otg.CurrentPosition[0];
      ProbeY := _otg.CurrentPosition[1];
      
      IF _otg.State = Struckig.TrajectoryState.Error
      THEN
        AbortErrorId(_otg.ErrorCode(), 'Trajectory Error');
      ELSIF _otg.State = Struckig.TrajectoryState.Idle
      THEN
        IF _splineIndex < 7
        THEN
          _splineIndex := _splineIndex + 1;
          _step.RepeatStep();
        ELSE
          _step.SetNext(ScriblyStep.AutomaticMovePenUp);                  
				END_IF
			END_IF      
    
    (* -------------------------------------------------------------------------------------------------------------------------------- *)
    ScriblyStep.AutomaticEnd:
    (* -------------------------------------------------------------------------------------------------------------------------------- *)
      SetBusy(FALSE);
  
  ELSE
    Abort('sequence contains unhandled step');
  END_CASE
UNTIL _step.IsNotRepeatable() OR_ELSE NOT Busy END_REPEAT

END_FUNCTION_BLOCK

// ---- ZApp/Unit/Scribly/_States/ScriblySequenceStop.TcPOU
FUNCTION_BLOCK ScriblySequenceStop EXTENDS ScriblySequence IMPLEMENTS ZCore.ISequence
VAR
  _step : ZCore.Step(ScriblyStep.StopBegin, ScriblyStep.StopEnd);
  _timerSim : ZAux.Timer;
END_VAR

IF OnStart(_step) THEN
  ; // init custom sequence variables here ...
END_IF

REPEAT
  LogStep();

  CASE _step.Index OF
    (* -------------------------------------------------------------------------------------------------------------------------------- *)
    ScriblyStep.StopBegin:
    (* -------------------------------------------------------------------------------------------------------------------------------- *)
      IF _step.OnEntry()
      THEN
        _actuator.Pen.UpAsync(THIS^);
        _axis.AxisX.StopAsync(THIS^);
        _axis.AxisY.StopAsync(THIS^);
			END_IF
      
      Await3(_actuator.Pen, _axis.AxisX, _axis.AxisY, nextStep:=ScriblyStep.StopEnd);

    (* -------------------------------------------------------------------------------------------------------------------------------- *)
    ScriblyStep.StopEnd:
    (* -------------------------------------------------------------------------------------------------------------------------------- *)    
      SetBusy(FALSE);
  
  ELSE
    Abort('sequence contains unhandled step');
  END_CASE
UNTIL _step.IsNotRepeatable() OR_ELSE NOT Busy END_REPEAT

END_FUNCTION_BLOCK

// ---- ZApp/Unit/Scribly/_States/ScriblySequenceGoHome.TcPOU
FUNCTION_BLOCK ScriblySequenceGoHome EXTENDS ScriblySequence IMPLEMENTS ZCore.ISequence
VAR
  _step : ZCore.Step(ScriblyStep.GohomeBegin, ScriblyStep.GohomeEnd);
  _timer : ZAux.Timer;
END_VAR

IF NOT Busy THEN
  RETURN;
END_IF

IF OnStart(_step) THEN
  ; // init custom sequence variables here ...
END_IF

IF OnStop() THEN
  RETURN; // external stop was triggered
END_IF

IF OnHalt() THEN
  ; // Halting := TRUE; // Uncomment to acknowledge that the sequence is halting
END_IF

REPEAT
  LogStep();

  CASE _step.Index OF
    (* -------------------------------------------------------------------------------------------------------------------------------- *)
    ScriblyStep.GoHomeBegin:
    (* -------------------------------------------------------------------------------------------------------------------------------- *)
      IF _step.OnEntry()
      THEN
        ;
			END_IF

      _step.SetNext(index:=ScriblyStep.GoHomeMoveUp);

    (* -------------------------------------------------------------------------------------------------------------------------------- *)
    ScriblyStep.GoHomeMoveUp:
    (* -------------------------------------------------------------------------------------------------------------------------------- *)
      IF _step.OnEntry()
      THEN
        _actuator.Pen.UpAsync(THIS^);
			END_IF
      
      Await(_actuator.Pen, nextStep:=ScriblyStep.GoHomeReferenceXY);

    (* -------------------------------------------------------------------------------------------------------------------------------- *)
    ScriblyStep.GoHomeReferenceXY:
    (* -------------------------------------------------------------------------------------------------------------------------------- *)
      IF _step.OnEntry()
      THEN
        _axis.AxisX.HomingAsync(THIS^);
        _axis.AxisY.HomingAsync(THIS^);
			END_IF
      
      Await3(_actuator.Pen, _axis.AxisX, _axis.AxisY, nextStep:=ScriblyStep.GoHomeEnd);

    (* -------------------------------------------------------------------------------------------------------------------------------- *)
    ScriblyStep.GoHomeEnd:
    (* -------------------------------------------------------------------------------------------------------------------------------- *)
      SetBusy(FALSE);
  
  ELSE
    Abort('sequence contains unhandled step');
  END_CASE
UNTIL _step.IsNotRepeatable() OR_ELSE NOT Busy END_REPEAT

END_FUNCTION_BLOCK

// ---- ZApp/Unit/Scribly/_States/ScriblySequenceFaultReaction.TcPOU
FUNCTION_BLOCK ScriblySequenceFaultReaction EXTENDS ScriblySequence IMPLEMENTS ZCore.ISequence
VAR
  _step : ZCore.Step(ScriblyStep.FaultReactionBegin, ScriblyStep.FaultReactionEnd);
  _timer : ZAux.Timer;
END_VAR

IF OnStart(_step) THEN
  ; // init custom sequence variables here ...
END_IF

REPEAT
  LogStep();

  CASE _step.Index OF
    (* -------------------------------------------------------------------------------------------------------------------------------- *)
    ScriblyStep.FaultReactionBegin:
    (* -------------------------------------------------------------------------------------------------------------------------------- *)
      IF _step.OnEntry()
      THEN
        _actuator.Pen.UpAsync(THIS^);
        _axis.AxisX.StopAsync(THIS^);
        _axis.AxisY.StopAsync(THIS^);
        _timer.WaitAsync(2);
			END_IF
      
      Await3(_actuator.Pen, _axis.AxisX, _axis.AxisY, nextStep:=ScriblyStep.FaultReactionEnd);
      IF _timer.Done
      THEN
        _step.SetNext(ScriblyStep.FaultReactionEnd);
			END_IF

    (* -------------------------------------------------------------------------------------------------------------------------------- *)
    ScriblyStep.FaultReactionEnd:
    (* -------------------------------------------------------------------------------------------------------------------------------- *)    
      SetBusy(FALSE);
  
  ELSE
    Abort('sequence contains unhandled step');
  END_CASE
UNTIL _step.IsNotRepeatable() OR_ELSE NOT Busy END_REPEAT

END_FUNCTION_BLOCK

// ---- ZApp/Unit/Scribly/ScriblyUnitProgram.TcPOU
/// each unit can run in its own PROGRAM and Task, respectively. However, this is optional and one may also
/// instantiate the unit in the ModuleProgram.
/// In order to keep initialization to a minimum, all ModuleContext objects that are required by the Unit are
/// given as FB_init parameter. These objects are
/// * data structs
/// * communication structs
/// * busmaster(s)
/// A unit should always be a root object (no parent) if it is running in its own context. If it runs in the same
/// task as the Module the parent may be set to the Module's Application.
PROGRAM ScriblyUnitProgram
VAR
{region "Scribly"}
{undefine RunInSeparateProgram}
{IF NOT (defined (Scribly_disabled)) AND (defined (RunInSeparateProgram))}
  Scribly : ScriblyUnit(name := 'Scribly', // name of the unit (for logging)
					  parent := 0, // caller of the Unit's cyclic method. If the Unit runs in its own context use 0
						configdata := ZGlobal.Data.Config.Scribly,
						machinedata := ZGlobal.Data.Machine.Scribly,
						calibrationdata := ZGlobal.Data.Calibration.Scribly,
						com := ZGlobal.Com.Unit.Scribly);
  {attribute 'section' := '__ZwPlcUnitProgramDeclaration__'}
  {attribute 'ZId' := '61e5b130-0fef-4d8b-85dd-afb1efcde47c'}
{END_IF}
{endregion}
{attribute '__ZwPlcUnitProgramDeclaration__'} // Do not remove this attribute! It is used for code generation.
END_VAR

// run the unit - the cylics of all children will be called as well

{region "Scribly"}
{undefine RunInSeparateProgram}
{IF NOT (defined (Scribly_disabled)) AND (defined (RunInSeparateProgram))}
  Scribly.Cyclic();
  {attribute 'section' := '__ZwPlcUnitProgramImplementation__'}
  {attribute 'ZId' := '61e5b130-0fef-4d8b-85dd-afb1efcde47c'}
{END_IF}
{endregion}
{attribute '__ZwPlcUnitProgramImplementation__'} // Do not remove this attribute! It is used for code generation.

END_PROGRAM
